PROGRAM MAIN
VAR
END_VAR

Q10();

END_PROGRAM

(* stored: Version 1.1.0.1, ProductVersion 3.1.4024.12
   POU MAIN: Id {df797fdd-9deb-4ee9-8b6c-571e8e3b10a2}, SpecialFunc None *)
